# EPICS substitutions: db/EL2042.substitutions
file EL2042.template
{ 	pattern
	{
		TERMINAL,
		DESC1,	ZNAM1,	ONAM1,	PINI1,
		DESC2,	ZNAM2,	ONAM2,	PINI2
	}
	{
	}
}
